# B&R Automation Studio project trace
Automation Studio 4.3.6.57 SP

## Configuration Config1

CPU PC_any, AutomationRuntime G4.34, Build 4.1.2, Vc V4.34.3

### Task classes (Cpu.sw)
```
Cyclic#1:
  sgenerator <- SampleData.sgenerator.prg
  datatrace <- DataTrace.datatrace.prg
Cyclic#8 (cycle 10000 us):
  savetrace <- DataTrace.savetrace.prg
Binaries: udbdef, TCData, sysconf, Role, User, iomap, ashwd, asfw, arconfig, ashwac
Libraries: FileIO, runtime, AsBrStr, astime, asieccon
```

### Hardware
```
PC : PC_any v1.1.0.0 (OrderNumber=PC)
  ConfigurationID = trace_Config1
  VolatileGlobalPvSize = 256000
  Cyclic8Duration = 10000
  FileDevice1
  FileDeviceName1 = CF
  FileDevicePath1 = C:\temp
```

## Logical view

Binary libraries used (declarations not repeated): operator, runtime, astime, AsIecCon, FileIO, AsBrStr


### Program Logical/SampleData/sgenerator (IEC)

#### Cyclic.st - Cyclic code
```iecst
PROGRAM _CYCLIC
	t:= t + 0.1;
	IF t > (24*3600.0) THEN
		t := 0;
	END_IF

	signal1 := 10*SIN(2*3.1415927*t);

	signal2 := signal2 + 1;
	IF signal2 > 10 THEN
		signal2 := -10;
		signal3 := -signal3;
	END_IF

	(* write data to trace *)
	g_dataTrace.currentRecord.real[0] := signal1;
	g_dataTrace.currentRecord.real[1] := signal2;
	g_dataTrace.currentRecord.real[2] := signal3;

END_PROGRAM
```

#### Init.st - Init code
```iecst
PROGRAM _INIT
	(* Insert code here *)
	 signal3 := 10.0;

	 g_dataTrace.enable := TRUE;
	 (* if g_dataTrace.enable is set to FALSE, data trace will stop and write data to CSV *)
END_PROGRAM
```

#### Variables.var - Local variables
```iecst
VAR
	signal1 : REAL;
	signal3 : REAL;
	signal2 : REAL;
	t : LREAL;
END_VAR
```

### TraceData.typ
```iecst
TYPE
	DataTrace_Typ : 	STRUCT
		enable : BOOL;
		currentWriteIndex : UDINT;
		currentReadIndex : USINT;
		elementsInTrace : UDINT;
		status : UINT;
		currentRecord : DataTraceRecord_Typ;
	END_STRUCT;
	DataTraceRecord_Typ : 	STRUCT
		real : ARRAY[0..g_MAX_DATA_TRACE_VARNUM_MINUS1]OF REAL;
	END_STRUCT;
END_TYPE
```

### TraceData.var
```iecst
VAR
	g_DATA_TRACE_FILEDEVICE : STRING[80] := 'CF';
END_VAR
VAR CONSTANT
	g_dataTraceColumns : ARRAY[0..g_MAX_DATA_TRACE_VARNUM_MINUS1] OF STRING[20] := ['signal1','signal2','signal3'];
END_VAR
VAR
	g_dataTrace : DataTrace_Typ;
END_VAR
VAR CONSTANT
	g_MAX_DATA_TRACE_RECORDS : UINT := 500; (* number of stored plc cycles (= rows)*)
	g_MAX_DATA_TRACE_VARNUM_MINUS1 : USINT := 2;  (* number of columns - 1 *)
END_VAR
VAR
	g_dataTraceRecords : ARRAY[0..g_MAX_DATA_TRACE_RECORDS] OF DataTraceRecord_Typ;
END_VAR
```

### Program Logical/DataTrace/datatrace (ANSIC)

#### Cyclic.c - Cyclic code
```c
/* ---------------------------------------------------------------------------------

simple data trace - execute this task in TC#1

visualize data e.g. with http://www.datplot.com/

------------------------------------------------------------------------------------ */
#include <bur/plctypes.h>
#include <string.h>

#ifdef _DEFAULT_INCLUDES
	#include <AsDefault.h>
#endif

void _CYCLIC ProgramCyclic(void)
{
	if( g_dataTrace.enable )
	{
		memcpy( &g_dataTraceRecords[g_dataTrace.currentWriteIndex], &g_dataTrace.currentRecord, sizeof(g_dataTraceRecords[0]) );

		if( ++g_dataTrace.elementsInTrace >= g_MAX_DATA_TRACE_RECORDS )
			g_dataTrace.elementsInTrace = g_MAX_DATA_TRACE_RECORDS;

		if( ++g_dataTrace.currentWriteIndex >= g_MAX_DATA_TRACE_RECORDS )
		{
			g_dataTrace.currentWriteIndex = 0;
			if( ++g_dataTrace.currentReadIndex >= g_MAX_DATA_TRACE_RECORDS )
				g_dataTrace.currentReadIndex = 0;
		}
	}
	else
	{

	}
}
```

#### Init.c - Initialization code
```c
#include <bur/plctypes.h>

#ifdef _DEFAULT_INCLUDES
	#include <AsDefault.h>
#endif

void _INIT ProgramInit(void)
{

}
```

#### Init.cpp - not listed in the package file held
```cpp
#include <bur/plctypes.h>

#ifdef _DEFAULT_INCLUDES
	#include <AsDefault.h>
#endif

unsigned long bur_heap_size = 0x10000;

void _INIT ProgramInit(void)
{

}
```

### Program Logical/DataTrace/savetrace (ANSIC)

#### ossupp.c
```c
#include <sys/types.h>
#include <sys/stat.h>

char heap[1000];
char *heapstart=heap;
char *heapend=&heap[1000];

void abort(void)
{
}

int fstat(int file, struct stat *st) {
  st->st_mode = S_IFCHR;
  return 0;
}

int close(int file){
    return -1;
}

int lseek(int file, int ptr, int dir){
    return 0;
}

int read(int file, char *ptr, int len){
    return 0;
}
int isatty(int file){
   return 1;
}

int writechar(char a)
{
	return 0;
}

int write(int file, char *ptr, int len){
    int todo;

    for (todo = 0; todo < len; todo++) {
        writechar(*ptr++);
    }
    return len;
}

caddr_t sbrk(int incr){
  static char *heap_end;
  char *prev_heap_end;

  if (heap_end == 0) {
    heap_end = heapstart;
  }
  prev_heap_end = heap_end;
  if (heap_end + incr > heapend)
    {
/*      _write (1, "Heap and stack collision\n", 25);*/
      abort ();
    }

  heap_end += incr;
  return (caddr_t) prev_heap_end;
}
```

#### Cyclic.c - Cyclic code
```c
/* ---------------------------------------------------------------------------------

simple data trace - execute this task in low priority task e.g. TC#8

visualize data e.g. with http://www.datplot.com/

------------------------------------------------------------------------------------ */
#include <bur/plctypes.h>
#include <stdio.h>
#include <string.h>

#ifdef _DEFAULT_INCLUDES
	#include <AsDefault.h>
#endif

#define BUFSIZE					65536

#define W_COMMAND 				0
#define GET_DATE_AND_TIME 		10
#define CREATE_FILE				20
#define WRITE_HEADER 			30
#define WRITE_RECORDS			40
#define WRITE_TO_FILE			50
#define CLOSE_FILE				60
#define RESET_DATA				70

char buffer[BUFSIZE];
char row[2048];
int i,n,j;
int len;

void _CYCLIC ProgramCyclic(void)
{

	switch( step )
	{
		case W_COMMAND:
		if( !g_dataTrace.enable && enableOld )
		{
			int i;
			int n = strlen(fileNamePrefix);
			if( n == 0 )
				strcpy( fileNamePrefix, "Trace" );
			/* replace invalid characters which are not allowed in file system */
			for( i = 0; i < n; ++i )
			{
				if( fileNamePrefix[i] < ' ' )
					fileNamePrefix[i] = ' ';
				switch( fileNamePrefix[i] )
				{
					case '\\': fileNamePrefix[i] = '_'; break;
					case '/': fileNamePrefix[i] = '_'; break;
				}
			}
			step = GET_DATE_AND_TIME;
		}
		enableOld = g_dataTrace.enable;
		break;

		case GET_DATE_AND_TIME:
		DTStructureGetTime(&fbGetTime);
		if( fbGetTime.status == 0 )
		{
			sprintf( fileName, "%s_%4.4u-%2.2u-%2.2u__%2.2u-%2.2u-%2.2u-%3.3u.csv",
				fileNamePrefix,
				dtStructure.year, dtStructure.month, dtStructure.day,
				dtStructure.hour, dtStructure.minute, dtStructure.second, dtStructure.millisec );
			step = CREATE_FILE;
		}
		break;

		case CREATE_FILE:
		fbFileCreate.enable = 1;
		fbFileCreate.pDevice = (UDINT) &g_DATA_TRACE_FILEDEVICE;
		fbFileCreate.pFile = (UDINT) fileName;
		FileCreate(&fbFileCreate);
		if( fbFileCreate.status == 0 )
		{
			fbFileWrite.enable = 1;
			fbFileWrite.ident = fbFileCreate.ident;
			fbFileWrite.offset = 0;

			fbFileClose.enable = 1;
			fbFileClose.ident = fbFileCreate.ident;
			step = WRITE_HEADER;
		}
		else if( fbFileCreate.status != 0xffff )
		{
			g_dataTrace.status = fbFileCreate.status;
			step = RESET_DATA;
		}
		break;

		case WRITE_HEADER:
		strcpy( row, "index" );
		for( n=0; n <= g_MAX_DATA_TRACE_VARNUM_MINUS1; ++n )
		{
			strcat( row, "," );
			strcat( row, g_dataTraceColumns[n] );
		}
		strcat( row, "\r\n" );

		fbFileWrite.pSrc = (UDINT) row;
		fbFileWrite.len = strlen(row);
		FileWrite( &fbFileWrite );
		if( fbFileWrite.status == 0 )
		{
			step = WRITE_RECORDS;
			fbFileWrite.offset += fbFileWrite.len;
		}
		else if( fbFileWrite.status != 0xffff )
		{
			step = W_COMMAND;
		}
		break;

		case WRITE_RECORDS:
		/* write to buffer first to increase speed */
		i = 0;
		j = 0;
		memset( buffer, 0, sizeof(buffer) );
		do
		{
			char tempstring[256];
			record = &g_dataTraceRecords[g_dataTrace.currentReadIndex];

			brsitoa( j, (UDINT) tempstring );
			strcpy( row, tempstring );
			for( n=0; n <= g_MAX_DATA_TRACE_VARNUM_MINUS1; ++n )
			{
				strcat( row, "," );
				brsftoa( record->real[n], (UDINT) tempstring );
				strcat( row, tempstring );
			}
			strcat( row, "\r\n" );
			len = n = strlen(row);
			strcpy( &buffer[i], row );
			i+= len;

			if( ++g_dataTrace.currentReadIndex >=  g_MAX_DATA_TRACE_RECORDS )
				g_dataTrace.currentReadIndex = 0;
			if( g_dataTrace.elementsInTrace )
				--g_dataTrace.elementsInTrace;
			++j;
		} while( (i < BUFSIZE) && (g_dataTrace.elementsInTrace) );
		fbFileWrite.pSrc = (UDINT) buffer;
		fbFileWrite.len = strlen(buffer);
		step = WRITE_TO_FILE;
		break;

		case WRITE_TO_FILE:
		/* write buffer to file */
		FileWrite( &fbFileWrite );
		if( fbFileWrite.status == 0 )
		{
			step = CLOSE_FILE;
		}
		else if( fbFileWrite.status != 0xffff )
		{
			g_dataTrace.status = fbFileWrite.status;
			step = RESET_DATA;
		}
		break;

		case CLOSE_FILE:
		FileClose( &fbFileClose );
		if( fbFileClose.status == 0 )
		{
			g_dataTrace.status = 0;
			step = RESET_DATA;
		}
		else if( fbFileClose.status != 0xffff )
		{
			g_dataTrace.status = fbFileClose.status;
			step = RESET_DATA;
		}
		break;

		case RESET_DATA:
		g_dataTrace.currentWriteIndex = 0;
		g_dataTrace.currentReadIndex = 0;
		g_dataTrace.currentReadIndex = 0;
		g_dataTrace.elementsInTrace = 0;
		step = W_COMMAND;
		break;

	}

}
```

#### Init.c - Initialization code
```c
#include <bur/plctypes.h>

#ifdef _DEFAULT_INCLUDES
	#include <AsDefault.h>
#endif
#include <string.h>
#include <math.h>

UDINT pNames[2];

void _INIT ProgramInit(void)
{

	fbGetTime.enable = 1;
	fbGetTime.pDTStructure = (UDINT) &dtStructure;
	step = 0;

	strcpy( fileNamePrefix, "Trace" );

	/* Defaultwerte */

}
```

#### Types.typ - Local data types
```iecst
TYPE
	ForceScaling : 	STRUCT
		offsetInkrements : INT;
		factorInkrements : INT;
		factorNewton : LREAL;
		currentInkrements : INT;
		currentForce : LREAL;
		forceMax : LREAL;
		cmdStoreOffset : USINT;
		enableForceMaximumCalc : BOOL;
	END_STRUCT;
END_TYPE
```

#### Variables.var - Local variables
```iecst
VAR
	enableOld : BOOL;
	step : UINT := 0;
	fileName : STRING[255] := '';
	fileNamePrefix : STRING[20] := '';
	record : REFERENCE TO DataTraceRecord_Typ;
	fbGetTime : DTStructureGetTime := (0);
	dtStructure : DTStructure := (0);
	fbFileClose : FileClose := (0);
	fbFileWrite : FileWrite := (0);
	fbFileCreate : FileCreate := (0);
END_VAR
```

#### Exit.cpp - not listed in the package file held
```cpp
#include <bur/plctypes.h>

#ifdef _DEFAULT_INCLUDES
	#include <AsDefault.h>
#endif

void _EXIT ProgramExit(void)
{

}
```

#### Init.cpp - not listed in the package file held
```cpp
#include <bur/plctypes.h>

#ifdef _DEFAULT_INCLUDES
	#include <AsDefault.h>
#endif
#include <string.h>
#include <math.h>

UDINT pNames[2];
unsigned long bur_heap_size = 0x10000;

void _INIT ProgramInit(void)
{

	fbGetTime.enable = 1;
	fbGetTime.pDTStructure = (UDINT) &dtStructure;
	step = 0;

	strcpy( fileNamePrefix, "Trace" );

	/* Defaultwerte */

}
```

Listed in the project but not available here: Logical/Global.typ, Logical/Global.var, Logical/SampleData/sgenerator/Exit.st, Logical/SampleData/sgenerator/Types.typ, Logical/DataTrace/datatrace/Exit.c, Logical/DataTrace/datatrace/Types.typ, Logical/DataTrace/datatrace/Variables.var, Logical/DataTrace/savetrace/Exit.c
